{attribute 'OPC.UA.DA.StructuredType' := '1'}
FUNCTION_BLOCK FB_Sensor_OceanControlsPressureTx_BVS006NA EXTENDS FB_BaseDevice IMPLEMENTS I_Device, I_Sensor
// This is a 0 to 6BAR pressure sensor from 4mA to 20mA

VAR

	{attribute 'OPC.UA.DA' := '0'} 
	eSensorType: E_SensorType;
	{attribute 'OPC.UA.DA' := '0'} 
	nRawInput AT %I*: INT;
	{attribute 'OPC.UA.DA' := '1'} 
	nCurrentValue: REAL;
	
	{attribute 'OPC.UA.DA' := '1'} 
	nVal4mA: REAL := 0; //kPA
	{attribute 'OPC.UA.DA' := '1'} 
	nVal20mA: REAL := 600; //kPA
	
END_VAR

calculate();

METHOD calculate : BOOL
VAR_INPUT
END_VAR
nCurrentValue := nVal4mA + (INT_TO_REAL(nRawInput) / GVL.nMaxADCOutput) * (nVal20mA - nVal4mA) ;
END_METHOD

{warning 'add method implementation '}
METHOD disable : BOOL
bEnable := FALSE;
END_METHOD

{warning 'add method implementation '}
METHOD enable : BOOL
bEnable := TRUE;
END_METHOD

{warning 'add method implementation '}
METHOD FB_init : BOOL
VAR_INPUT
	(* if TRUE, the retain variables are initialized (warm start / cold start)*)
	bInitRetains	: BOOL;
	(* if TRUE, the instance afterwards gets moved into the copy code (online change)*)
	bInCopyCode	: BOOL;
	SensorID	: STRING(80);
	SensorDescr	: STRING(255);
	SensorType	: E_SensorType;
	
END_VAR
sID := SensorID;
sDescr := SensorDescr;
eSensorType := SensorType;
END_METHOD

{warning 'add method implementation '}
METHOD getType : E_SensorType
getType := eSensorType;
END_METHOD

{warning 'add method implementation '}
METHOD getValue : REAL
getValue := nCurrentValue;
END_METHOD

METHOD setLimits : BOOL
VAR_INPUT
	Val_4mA: 	REAL;
	Val_20mA: 	REAL;
END_VAR
nVal4mA := Val_4mA;
nVal20mA := Val_20mA;
END_METHOD

{warning 'add method implementation '}
METHOD write : BOOL
END_METHOD

END_FUNCTION_BLOCK

(* stored: Version 1.1.0.1, ProductVersion 3.1.4024.12
   POU FB_Sensor_OceanControlsPressureTx_BVS006NA: Id {5eeff715-444e-40ae-8558-5ddf7f8fb826}, SpecialFunc None
   Method calculate: Id {918b74fa-5657-4007-8a25-d97f94782e14}
   Method disable: Id {ce35d87c-e1ce-4ef0-86a5-ef8420d2fd64}
   Method enable: Id {9e67d969-ab93-4658-99b0-833b5b915c82}
   Method FB_init: Id {06d31db5-7880-4457-8fe8-d151c58862c3}
   Method getType: Id {8c43849d-c927-41d0-96cf-6c16fc0815a9}
   Method getValue: Id {5afbf4bb-e15b-4277-b764-b2e869e90722}
   Method setLimits: Id {c3022aee-f44f-486f-8fc7-f52de379b09c}
   Method write: Id {1e5211c2-b798-47e5-a6d4-8903204343ba} *)
